INTERFACE IAssertionListener

METHOD OnAssertionFailed
VAR_INPUT
    AssertionMessage : T_MaxString;
    ExpectedAsString : T_MaxString;
    ActualAsString   : T_MaxString;
END_VAR
END_METHOD

PROPERTY TestName : T_MaxString
GET
END_GET
END_PROPERTY

END_INTERFACE

(* stored: Version 1.1.0.1, ProductVersion 3.1.4024.4
   Itf IAssertionListener: Id {fe3d0b3b-5ee1-4fd7-bdd2-334821d13a4d}
   Method OnAssertionFailed: Id {d9aff967-7824-405f-9421-8751c88d368f}
   Property TestName: Id {07b43fbb-79b5-43a4-b4fa-0f3491665c38}
   Get Get: Id {d13fb6a0-d46d-436f-930f-e3b14b83aa81} *)
